FUNCTION_BLOCK MUX_ANY (* Abstract superclass for IEC 61131-3 multiplexers *)
  (* Standard: 61131-3 *)
  (* Version 0.0, 2004-12-15, JHC, Rockwell Automation, Converted from SRC format. *)
  (* Compiler header: package fb.rt.plc.select; *)
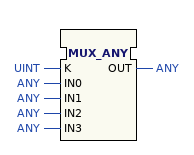
  VAR_INPUT
    K : UINT; (* Selector,0<=K<=3 *)
    IN0 : ANY; (* Output when K=0 *)
    IN1 : ANY; (* Output when K=1 *)
    IN2 : ANY; (* Output when K=2 *)
    IN3 : ANY; (* Output when K=3 *)
  END_VAR
  VAR_OUTPUT
    OUT : ANY;
  END_VAR
END_FUNCTION_BLOCK
